TYPE DUT_CheckCutterAlreadyPresentOnDrums :
STRUCT
	Id			: DINT;
	Drum		: STRING(30);
	Present		: DINT;
END_STRUCT
END_TYPE

(* stored: Version 1.1.0.1, ProductVersion 3.1.4024.15
   DUT DUT_CheckCutterAlreadyPresentOnDrums: Id {02e6a8c6-e41e-4317-a87b-2f6b1ed909fa} *)
